# EPICS substitutions: evrSupport/Db/evr/evrIMXX.substitutions
#==============================================================================
#
# Abs:  LCLS EVR IOC records for Current Monitor (IM) IOCs
#
# Name: evrIMXX.substitutions
#
#==============================================================================
#
file evr.db
{
#                           Default Pulse
#	 Device      Card   Delay   Width (clock ticks)
pattern { DEV      , CARD , DELAY , WIDTH }
	{ $(DEVICE),  0   ,   0   ,  12   }
}
#Note - there is a dependency on event code assignments and triggers.
#     When changing event code assignments below, also change the appropriate
#     IOC-*-IM*trig.substitutions file!
file evrEventCtrl.db
{
#	  Device      Card  <----------------------------  Event -------------------------->
pattern { DEV       , CARD , NAME    , ID ,P0,P1,P2,P3,P4,P5,P6,P7,P8,P9,P10,P11,P12,P13,VME}
	{ $(DEVICE) ,   0  , EVENT1  ,140 , 0, 0, 0, 0, 0, 0, 0, 0, 0, 0, 0 , 0 , 0 , 0 , 0 }
	{ $(DEVICE) ,   0  , EVENT2  , 50 , 0, 0, 0, 0, 0, 0, 0, 0, 0, 0, 0 , 0 , 1 , 1 , 0 }
	{ $(DEVICE) ,   0  , EVENT3  , 60 , 0, 0, 0, 0, 0, 0, 0, 0, 0, 0, 0 , 0 , 0 , 0 , 0 }
	{ $(DEVICE) ,   0  , EVENT4  , 40 , 0, 0, 0, 0, 0, 0, 0, 0, 0, 0, 0 , 0 , 0 , 0 , 0 }
	{ $(DEVICE) ,   0  , EVENT5  , 41 , 0, 0, 0, 0, 0, 0, 0, 0, 0, 0, 0 , 0 , 0 , 0 , 0 }
	{ $(DEVICE) ,   0  , EVENT6  , 42 , 1, 1, 1, 1, 1, 1, 1, 1, 1, 1, 1 , 1 , 0 , 0 , 0 }
	{ $(DEVICE) ,   0  , EVENT7  , 43 , 0, 0, 0, 0, 0, 0, 0, 0, 0, 0, 0 , 0 , 0 , 0 , 0 }
	{ $(DEVICE) ,   0  , EVENT8  , 44 , 0, 0, 0, 0, 0, 0, 0, 0, 0, 0, 0 , 0 , 0 , 0 , 0 }
	{ $(DEVICE) ,   0  , EVENT9  , 45 , 0, 0, 0, 0, 0, 0, 0, 0, 0, 0, 0 , 0 , 0 , 0 , 0 }
	{ $(DEVICE) ,   0  , EVENT10 , 46 , 0, 0, 0, 0, 0, 0, 0, 0, 0, 0, 0 , 0 , 0 , 0 , 0 }
	{ $(DEVICE) ,   0  , EVENT11 , 11 , 0, 0, 0, 0, 0, 0, 0, 0, 0, 0, 0 , 0 , 0 , 0 , 0 }
	{ $(DEVICE) ,   0  , EVENT12 , 12 , 0, 0, 0, 0, 0, 0, 0, 0, 0, 0, 0 , 0 , 0 , 0 , 0 }
	{ $(DEVICE) ,   0  , EVENT13 , 13 , 0, 0, 0, 0, 0, 0, 0, 0, 0, 0, 0 , 0 , 0 , 0 , 0 }
	{ $(DEVICE) ,   0  , EVENT14 , 14 , 0, 0, 0, 0, 0, 0, 0, 0, 0, 0, 0 , 0 , 0 , 0 , 0 }
}
